(* IEC 61131-3 sources: AXOpen/src/templates.simple/ax/src/templates/starterunit/DataManagers, 4 files *)

(* ---- FragmentsProcessDataManager.st ---- *)
NAMESPACE axosimple.StarterUnitTemplate
    USING axosimple;
    USING AXOpen.Data;
    USING AXOpen.Core;
    USING System.Strings;

    {S7.extern=ReadWrite}
    CLASS FragmentProcessDataManger
        EXTENDS AXOpen.Data.AxoDataExchange
        VAR PUBLIC
            {#ix-generic:TOnline}
            {#ix-generic:TPlain as POCO}
            {#ix-attr:[AXOpen.Data.AxoDataEntityAttribute]}
            {#ix-attr:[Container(Layout.Stack)]}
            {#ix-set:AttributeName = "<#StarterUnitTemplate#>"}
            Payload : ProcessData;
        END_VAR
    END_CLASS
END_NAMESPACE

(* ---- FragmentTechnologyDataManger.st ---- *)
NAMESPACE axosimple.StarterUnitTemplate
    USING axosimple;
    USING AXOpen.Data;
    USING AXOpen.Core;
    USING System.Strings;

    {S7.extern=ReadWrite}
    CLASS FragmentTechnologyDataManger
        EXTENDS AXOpen.Data.AxoDataExchange
        VAR PUBLIC
            {#ix-generic:TOnline}
            {#ix-generic:TPlain as POCO}
            {#ix-attr:[AXOpen.Data.AxoDataEntityAttribute]}
            {#ix-attr:[Container(Layout.Stack)]}
            {#ix-set:AttributeName = "<#UnitTemplate#>"}
            Payload : axosimple.StarterUnitTemplate.TechnologyData;
        END_VAR
    END_CLASS
END_NAMESPACE

(* ---- ProcessDataManger.st ---- *)
NAMESPACE axosimple.StarterUnitTemplate
    USING axosimple;
    USING AXOpen.Data;
    USING AXOpen.Core;
    USING System.Strings;

    {S7.extern=ReadWrite}
    CLASS ProcessDataManager
        EXTENDS AXOpen.Data.AxoDataFragmentExchange
        VAR PUBLIC
            {#ix-attr:[AXOpen.Data.AxoDataFragmentAttribute]}
            Shared : axosimple.EntityHeaderDataManager;
            {#ix-attr:[AXOpen.Data.AxoDataFragmentAttribute]}
            DataManger : axosimple.StarterUnitTemplate.FragmentProcessDataManger;
        END_VAR
    END_CLASS
END_NAMESPACE

(* ---- TechnologyDataManager.st ---- *)
NAMESPACE axosimple.StarterUnitTemplate
    USING axosimple;
    USING AXOpen.Data;
    USING AXOpen.Core;
    USING System.Strings;

    CLASS TechnologyDataManager
        EXTENDS AXOpen.Data.AxoDataFragmentExchange
        VAR PUBLIC
            {#ix-attr:[AXOpen.Data.AxoDataFragmentAttribute]}
            Shared : TechnologyCommonDataManager;

            {#ix-attr:[AXOpen.Data.AxoDataFragmentAttribute]}
            DataManger : FragmentTechnologyDataManger;
        END_VAR
    END_CLASS
END_NAMESPACE
